INTERFACE ILimitedStringBuilder

METHOD  Append : IStringBuilder // Append text to t current build string.
VAR_INPUT
	Text : STRING(GVL_Param_AUT_Utilities.StringBuilder_MaxStringLength); //Text to append to current build string
END_VAR
END_METHOD

METHOD  AppendWithFormat : IStringBuilder // Append text to t current build string.
VAR_INPUT
	Value : ANY;    //T_Arg; // Value to format
	Format : STRING(GVL_Param_AUT_Utilities.StringBuilder_MaxStringLength); // Format to apply 
END_VAR
END_METHOD

METHOD Reset : ILimitedStringBuilder //Reset current build string to an empty string.
END_METHOD

METHOD ToString : STRING(GVL_Param_AUT_Utilities.StringBuilder_MaxStringLength)    //Returns current build string.
END_METHOD

METHOD ToWString : WSTRING(GVL_Param_AUT_Utilities.StringBuilder_MaxStringLength) //Returns current build string.
END_METHOD

END_INTERFACE

(* stored: Version 1.1.0.1
   Itf ILimitedStringBuilder: Id {3b3cc063-dd61-45f7-aa02-e6f092d65ebb}
   Method Append: Id {cb85310e-4987-4cc7-8a05-9832a0be426b}
   Method AppendWithFormat: Id {dabae837-2235-48b2-a5a9-95583277cf7a}
   Method Reset: Id {ebe76031-5bda-45af-a5b1-6f04a5768308}
   Method ToString: Id {5e66f779-8a90-4f31-b710-213cc3abfd38}
   Method ToWString: Id {9fa4eae6-5cd2-4dcf-a3e4-15e1a138eff3} *)
